FUNCTION_BLOCK Station EXTENDS Objective
VAR
	
	{attribute 'hide'}
	Position			: LREAL;

END_VAR

{attribute 'monitoring' := 'variable'}
PROPERTY CurrentMover : REFERENCE TO Mover
GET
VAR
	
	i: USINT;	
	difference: LREAL;
	
END_VAR

// default to unassigned
CurrentMover REF= 0;

FOR i := 0 TO SIZEOF( internalTrackedMovers ) / SIZEOF( internalTrackedMovers[0] ) - 1 DO
	
	// In order to deal with the rollover, we need to evaluate distance between congruence classes
	// e.g. On a 4m track, if the Station is at 0.34mm and the Mover is at 3999.8mm, then this is considered 'in position'	

	IF internalTrackedMovers[i] <> 0 THEN
		
		// difference	:= ABS( MODABS( TrackedMovers[i]^.AxisReference.NcToPlc.ActPos,GVL.TRACK_LENGTH ) - THIS^.TrackPosition );
		difference	:= ABS( internalTrackedMovers[i]^.AxisReference.NcToPlc.ModuloActPos - TrackPosition );
		
		IF MIN( difference, GVL.TRACK_LENGTH - difference ) < 1.0 AND NOT internalTrackedMovers[i]^.Busy THEN
			CurrentMover	REF= internalTrackedMovers[i]^;
		END_IF
	END_IF

END_FOR
END_GET
END_PROPERTY

METHOD Cyclic : BOOL

VAR
	i: USINT;
END_VAR


FOR i := 0 TO GVL.NUM_MOVERS - 1 DO
	
	// This mover is no longer destined for any station
	IF internalTrackedMovers[i] <> 0 AND_THEN internalTrackedMovers[i]^.CurrentMoveType <> MOVETYPE_STATION THEN
		internalTrackedMovers[i]	:= 0;
	// This mover is no longer destined for this specific station. Comparing instance path seems to be the best way to do this comparison?
	ELSIF internalTrackedMovers[i] <> 0 AND_THEN internalTrackedMovers[i]^.CurrentObjective <> InstancePath THEN
		internalTrackedMovers[i]	:= 0;
	END_IF

END_FOR
END_METHOD

{attribute 'monitoring' := 'variable'}
PROPERTY MoverInPosition : BOOL
GET
VAR
	
	i		: USINT;	
	difference: LREAL;
	
END_VAR

// default to false
MoverInPosition		:= FALSE;

FOR i := 0 TO SIZEOF( internalTrackedMovers ) / SIZEOF( internalTrackedMovers[0] ) - 1 DO
	
	// In order to deal with the rollover, we need to evaluate distance between congruence classes
	// e.g. On a 4m track, if the Station is at 0.34 mm and the Mover is at 3999.8mm, then this is considered 'in position' 
	
	// todo: make in-position tolerance adjustable. add condition that mover is stopped?
	IF internalTrackedMovers[i] <> 0 THEN
		difference	:= ABS( MODABS( internalTrackedMovers[i]^.AxisReference.NcToPlc.ActPos,GVL.TRACK_LENGTH ) - THIS^.TrackPosition );
      IF (MIN( difference, GVL.TRACK_LENGTH - difference ) < 1.0 ) AND NOT internalTrackedMovers[i]^.Busy THEN
			MoverInPosition		:= TRUE;
		END_IF
 	END_IF;

END_FOR
END_GET
END_PROPERTY

{attribute 'monitoring' := 'call'}
PROPERTY TrackPosition : LREAL
GET


	TrackPosition		:= Position;
END_GET
SET


	Position		:= TrackPosition;
END_SET
END_PROPERTY

END_FUNCTION_BLOCK

(* stored: Version 1.1.0.1, ProductVersion 3.1.4024.9
   POU Station: Id {5b67f0b3-4286-49f2-9b21-1e637f521584}, SpecialFunc None
   Folder Methods: Id {b783a2bf-4b7a-4aa5-9ae9-11ae8e9caf95}
   Folder Properties: Id {a0c9a439-1ed2-41be-8a26-9d0fb905bf29}
   Property CurrentMover: Id {4e639a8f-b6e4-4381-9171-31b76bf41c77}
   Get Get: Id {590174cc-2a32-4e82-86cf-1c2eff136812}
   Method Cyclic: Id {b1387964-723e-4a2a-a4b6-2d82b2e2e3a7}
   Property MoverInPosition: Id {7b7104e7-1816-4b78-b1aa-ded30e5ff809}
   Get Get: Id {11118b5e-d8b3-4427-a8f3-470e1381cae5}
   Property TrackPosition: Id {a036a85b-a6ff-4e53-924d-8183c40c2111}
   Get Get: Id {9b1fb402-d994-4b37-826c-4ff94e3f9cbc}
   Set Set: Id {6983000b-95aa-45e5-9d08-48de77decd80} *)
